// TwinCAT 3 PLC project main
// libraries:
//   Tc2_Math, * (Beckhoff Automation GmbH)
//   Tc2_MC2, * (Beckhoff Automation GmbH)
//   Tc2_Standard, * (Beckhoff Automation GmbH)
//   Tc2_System, * (Beckhoff Automation GmbH)
//   Tc3_Module, * (Beckhoff Automation GmbH)
//   VisuDialogs, * (System)
// project tree:
//   Global Variables/ Global_Variables.TcGVL, Variable_Configuration.TcGVL
//   / GlobalImagePool.TcGIPO (not stored), Standard.TcTTO, 视图管理器.TcVMO (not stored)
//   POUs/ AxisWriteParameter.TcPOU, Axis_Limit_Stop.TcPOU, Axis_Move.TcPOU, Axis_Power.TcPOU, Axis_stop.TcPOU, Axis_To_Zero.TcPOU, BackwardWindingStart.TcPOU, BLINK.TcPOU, ForwardWindingStart.TcPOU, MAIN.TcPOU, MainAxisRot.TcPOU, Manual_Left.TcPOU, Manual_Right.TcPOU, Motor_Init.TcPOU, Pulse2.TcPOU, ReadEncSpeed.TcPOU
//   Visualizations/ HMI1.TcVIS
// real-time tasks:
//   TASK Standard: cycle T#10ms, priority 20, ADS port 350
// motion (NC):
//   TASK NC-Task 1 SAF: cycle T#2ms, priority 4, ADS port 501
//   TASK NC-Task 1 SVB: cycle T#10ms, priority 8, ADS port 511
//   AXIS Axis 1 (id 1)
//     OtherSettings: AllowMotionCmdToSlave=true
//     encoder EncType=1
//       EncPara: ScaleFactorNumerator=0.00015625
//     drive DrvType=5
//       Analog: TorqueSetpointScale=10, ScaleFactorActTorque=0.1
//       TimeComp: TaskDelayCycles=1
//     controller CtrType=1
//       CtrPara: PriorControlFactor=1
//         Observer: BandWidth=20
//   AXIS Axis 2 (id 2)
//     OtherSettings: AllowMotionCmdToSlave=true
//     encoder EncType=4
//       EncPara: ScaleFactorNumerator=0.00025, MaxCount=#x0000ffff
//     drive DrvType=5
//       Analog: TorqueSetpointScale=10, ScaleFactorActTorque=0.1
//       TimeComp: TaskDelayCycles=1
//     controller CtrType=1
//       CtrPara: PriorControlFactor=1
//         Observer: BandWidth=20
//   AXIS Axis 3 (id 3)
//     OtherSettings: AllowMotionCmdToSlave=true
//     encoder EncType=1
//       EncPara: ScaleFactorNumerator=0.25
//     drive DrvType=5
//       Analog: TorqueSetpointScale=10, ScaleFactorActTorque=0.1
//       TimeComp: TaskDelayCycles=1
//     controller CtrType=1
//       CtrPara: PriorControlFactor=1
//         Observer: BandWidth=20
// variable links:
//   main/main Instance <-> NC-Task 1 SAF/Axes/Axis 1
//     Standard Inputs/.Axis1.NcToPlc <-> Outputs/ToPlc
//     Standard Outputs/.Axis1.PlcToNc <-> Inputs/FromPlc
//   main/main Instance <-> NC-Task 1 SAF/Axes/Axis 2
//     Standard Inputs/.Axis2.NcToPlc <-> Outputs/ToPlc
//     Standard Outputs/.Axis2.PlcToNc <-> Inputs/FromPlc
//   main/main Instance <-> NC-Task 1 SAF/Axes/Axis 3
//     Standard Inputs/.Axis3.NcToPlc <-> Outputs/ToPlc
//     Standard Outputs/.Axis3.PlcToNc <-> Inputs/FromPlc

CONFIGURATION main
    RESOURCE PLC ON TwinCAT3
        TASK Standard(INTERVAL := T#10ms, PRIORITY := 20);
        PROGRAM MAIN WITH Standard : MAIN;
    END_RESOURCE
END_CONFIGURATION

// ---- Global Variables/Global_Variables.TcGVL
{attribute 'Tc2GvlVarNames'}
VAR_GLOBAL
	Axis1: Axis_Ref;
	Axis2: Axis_Ref;
	Axis3: Axis_Ref;
END_VAR

// ---- Global Variables/Variable_Configuration.TcGVL
{attribute 'Tc2GvlVarNames'}
VAR_CONFIG
END_VAR

// ---- POUs/MAIN.TcPOU
PROGRAM MAIN
VAR_INPUT
	FootPedalPressed	AT%I*	:	BOOL;	(*主轴脚踏开关i1*)
	WireForwardWindingControl	AT%I*	:	BOOL;	(*自动排线正i2*)
	WireBackwardWindingControl	AT%I*	:	BOOL;	(*自动排线反i3*)
	MainAxisRotatingDirection AT%I*:	BOOL:= FALSE;	(*主轴旋转方向i4,TRUE 反向，FALSE正向*)
	MainAxisRotatingBackFlag: BOOL:= TRUE;
	cannel_5 AT%I*: BOOL;
	WireBackwardManualControl 	AT%I*	:	BOOL;	(*手动排线反i6*)
	WireForwardManualControl	AT%I*	:	BOOL;	(*手动排线正i7*)
	WireLeadPositiveLimit 	AT%I*	:	BOOL;	(*排线轴正限位i8*)
	WireLeadNegativeLimit 	AT%I*	:	BOOL;	(*排线轴负限位i9*)
	WireLeadToZero		AT%I*	:	BOOL;	(*排线轴寻零i10*)
	EL180911 AT%I*: BOOL;
	EL180912 AT%I*: BOOL;

	MainAxisSpeedControl	AT%I*	:	INT:=32767;		(*主轴调速, 模拟量*)

END_VAR
VAR_OUTPUT
	OpMode	AT%Q*: SINT:=8;	(*OP MODE*)
	Opmode2 AT%Q*: SINT:=8;	(*OP MODE*)

	status_Axis_forward		AT%Q*:	BOOL;	(*主轴正转o1*)
	status_Axis_backward		AT%Q*:	BOOL;	(*主轴反转o2*)
	Manual_control_forward	AT%Q*:	BOOL;	(*手动正转o3*)
	Manual_control_backward	AT%Q*:	BOOL;	(*手动反转o4*)
	Auto_control_forward		AT%Q*:	BOOL;	(*自动正转o5*)
	Auto_control_backward		AT%Q*:	BOOL;	(*自动反转o6*)
	Forward_position_limit		AT%Q*: 	BOOL;	(*起点限位o7*)
	Backward_position_limit	AT%Q*:	BOOL;	(*终点限位o8*)
	T510_X1		AT%Q*:	BOOL:=	FALSE;	(*T510的x1, 接主轴驱动器o9*)
	T510_X2		AT%Q*:	BOOL:=	FALSE;	(*T510的x2, 接主轴驱动器o10*)
	MotorEnable1 	AT%Q*:	BOOL:=	FALSE;	(*主轴电机使能o11*)
	MotorEnable2 	AT%Q*:	BOOL:=	FALSE;	(*主轴电机使能o12*)

END_VAR
VAR
	Flag1: BOOL;
	timer1: Pulse2;
	shanshuo: BLINK;

	AxisPower: Axis_Power;
	AxisReset2:MC_Reset;
	AxisReset1: MC_Reset;
	MoveVelPlus: MC_MoveVelocity;
	MoveVelDec: MC_MoveVelocity;
	absMove1: MC_MoveAbsolute;
	absMove2: MC_MoveAbsolute;

	MOTORINIT: Motor_Init;
	WriteParameter: AxisWriteParameter;
	AxisStop: Axis_Limit_Stop;
	AxisStop2: Axis_stop;
	AxisToZero:Axis_To_Zero;
	manleft:Manual_Left;
	manright			:	Manual_Right;
	AxisMove			:	Axis_Move;
	MainAxisRotation	:	MainAxisRot;
	ReadEncoderVel	:	ReadEncSpeed;
	WireWeights	:	REAL:=	2.4;
	TargetMainAxisSpeed	:	REAL:=	8;
	ManualControlVelocity	:	REAL:=	8;
	SlaveAxisBackZero	:	REAL:= 8;

END_VAR


(********************************************************  轴使能   ************************************************************)
AxisPower(
	SpeedControl:=MainAxisSpeedControl,
	Power_Status=> );
AxisReset1(
	Execute:=EL180911,
	Axis:= Axis1,
	Done=> ,
	Busy=> ,
	Error=> ,
	ErrorID=> );

AxisReset2(
	Execute:=EL180911,
	Axis:= Axis3,
	Done=> ,
	Busy=> ,
	Error=> ,
	ErrorID=> );

AxisStop(
	Execute_:=WireLeadPositiveLimit,
	Execute_2:=WireLeadNegativeLimit ,
	Decelerations:=1500,
	Flag1=>Forward_position_limit,
	Flag2=> Backward_position_limit);

ReadEncoderVel(input1:= AxisPower.Power_Status, RealSpeed=> );

(****************************************************  主轴旋转方向设定	********************************************************)
IF MainAxisRotatingDirection THEN
	MainAxisRotatingBackFlag:=FALSE;
	status_Axis_forward:=TRUE;
	status_Axis_backward:=FALSE;
ELSE
	MainAxisRotatingBackFlag:= TRUE;
	status_Axis_forward:=FALSE;
	status_Axis_backward:=TRUE;
END_IF

(******************************************************	正转向右启动	*******************************************************)
IF MainAxisRotatingDirection THEN
	IF FootPedalPressed THEN
			T510_X1:=TRUE;
			MOTORINIT(forward_start:=MainAxisRotatingDirection , backward_start:=T510_X1 , Flag=> MotorEnable1);
		ELSE
			T510_X1:=FALSE;
			MOTORINIT(forward_start:=FALSE , backward_start:=T510_X1 , Flag=> MotorEnable1);
	END_IF
	IF WireForwardWindingControl THEN
		IF FootPedalPressed THEN OpMode:=8;
		END_IF
	(*伺服动作*)
		MoveVelPlus(
				Execute:=FootPedalPressed ,
				Velocity:= (WireWeights*TargetMainAxisSpeed),
				Acceleration:= ,
				Deceleration:= ,
				Jerk:= ,
				Direction:= MC_Positive_Direction,
				BufferMode:= ,
				Options:= ,
				Axis:=Axis1 ,
				InVelocity=> ,
				Busy=> ,
				Active=>Auto_control_forward ,
				CommandAborted=> ,
				Error=> ,
				ErrorID=> );

		AxisStop2(Execute_:= FootPedalPressed);
		(*AxisMove(Input1:=FootPedalPressed );*)
	END_IF

	(*正向向左启动*)
	IF WireBackwardWindingControl THEN
		IF FootPedalPressed THEN OpMode:=8;
		END_IF
	(*私服动作*)
		MoveVelDec(
				Execute:= FootPedalPressed,
				Velocity:= (WireWeights*TargetMainAxisSpeed),
				Acceleration:= ,
				Deceleration:= ,
				Jerk:= ,
				Direction:= MC_Negative_Direction,
				BufferMode:= ,
				Options:= ,
				Axis:=Axis1 ,
				InVelocity=> ,
				Busy=> ,
				Active=>Auto_control_backward ,
				CommandAborted=> ,
				Error=> ,
				ErrorID=> );
		AxisStop2(Execute_:= FootPedalPressed);
	END_IF
END_IF


(*****************************************************	反转向右启动	******************************************************)
IF MainAxisRotatingBackFlag THEN
	IF FootPedalPressed THEN
			T510_X2:=TRUE;
			MOTORINIT(forward_start:=MainAxisRotatingBackFlag , backward_start:=T510_X2 , Flag=> MotorEnable1);
		ELSE
			T510_X2:=FALSE;
			MOTORINIT(
					forward_start:=FALSE ,
					backward_start:=T510_X2 ,
					Flag=> MotorEnable1);
	END_IF
	IF WireForwardWindingControl THEN
		IF FootPedalPressed THEN OpMode:=8;
		END_IF
		MoveVelPlus(
				Execute:=FootPedalPressed ,
				Velocity:= (WireWeights*TargetMainAxisSpeed),
				Acceleration:= ,
				Deceleration:= ,
				Jerk:= ,
				Direction:= MC_Positive_Direction,
				BufferMode:= ,
				Options:= ,
				Axis:=Axis1 ,
				InVelocity=> ,
				Busy=> ,
				Active=>Auto_control_forward ,
				CommandAborted=> ,
				Error=> ,
				ErrorID=> );
		AxisStop2(Execute_:= FootPedalPressed);
	END_IF

	(*反转向左启动*)
	IF WireBackwardWindingControl THEN
		MoveVelDec(
				Execute:= FootPedalPressed,
				Velocity:= (WireWeights*TargetMainAxisSpeed),
				Acceleration:= ,
				Deceleration:= ,
				Jerk:= ,
				Direction:= MC_Negative_Direction,
				BufferMode:= ,
				Options:= ,
				Axis:=Axis1 ,
				InVelocity=> ,
				Busy=> ,
				Active=>Auto_control_backward ,
				CommandAborted=> ,
				Error=> ,
				ErrorID=> );
		AxisStop2(Execute_:= FootPedalPressed);
	END_IF
END_IF


(*****************************************************	手动控制正向启动	************************************************************)
	(*私服动作*)
IF WireForwardManualControl THEN
	OpMode:=8;
END_IF
manleft(
	Input1:=	WireForwardManualControl,
	ManualCotrolSpeed	:=	ManualControlVelocity ,
	Flag1	=>	Manual_control_forward);

(*Flag1:=REAL_TO_INT(0.02432*MainAxisSpeedControl);
timer1(button1:= WireForwardManualControl, time_fuction:=Flag1, Flag=>status_Axis_forward );*)


(****************************************************	手动控制反向启动	************************************************************)
	(*私服动作*)
IF WireBackwardManualControl THEN
	OpMode:=8;
END_IF
manright(
	Input1:=WireBackwardManualControl,
	ManualCotrolSpeed	:=ManualControlVelocity ,
	Flag1=> Manual_control_backward);

(**********************************************************	排线轴归零	*********************************************************************)
IF WireLeadToZero THEN
	OpMode:=8;
END_IF
AxisToZero(
	Flag:= WireLeadToZero,
	BackZeroSpeed:=SlaveAxisBackZero);

(**********************************************************	主轴旋转控制	*****************************************************************)
IF FootPedalPressed THEN
	OpMode2:=8;
END_IF
MainAxisRotation(
	Input1:=FootPedalPressed,
	ForwardRotFlag:=MainAxisRotatingDirection,
	BackwardRotFlag:=MainAxisRotatingBackFlag,
	InputTargetSpeed:= TargetMainAxisSpeed);

END_PROGRAM

// ---- POUs/Pulse2.TcPOU
FUNCTION_BLOCK Pulse2
VAR_INPUT
	button1: BOOL;
	time_fuction: INT;
END_VAR
VAR_OUTPUT
	Flag: BOOL;
END_VAR
VAR
	Timer1: TON;
END_VAR

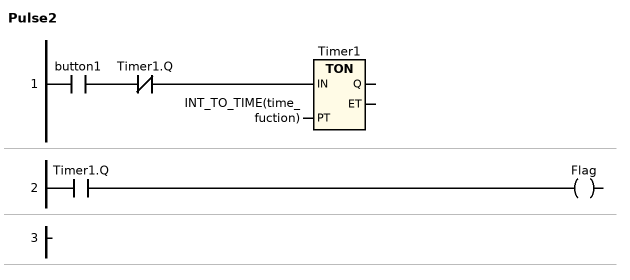
// NETWORK 1
Timer1(IN := button1 AND NOT Timer1.Q, PT := INT_TO_TIME(time_fuction)); // TON

// NETWORK 2
Flag := Timer1.Q;

// NETWORK 3

END_FUNCTION_BLOCK

// ---- POUs/BLINK.TcPOU
FUNCTION_BLOCK BLINK
VAR_INPUT
	ENABLE: BOOL;
END_VAR
VAR_OUTPUT
	OUT: BOOL;
END_VAR
VAR
	TIMELOW: INT;
	TIMEHIGH: INT;
	T37: TON;
	T38: TOF;
	TEMP1: BOOL;
END_VAR

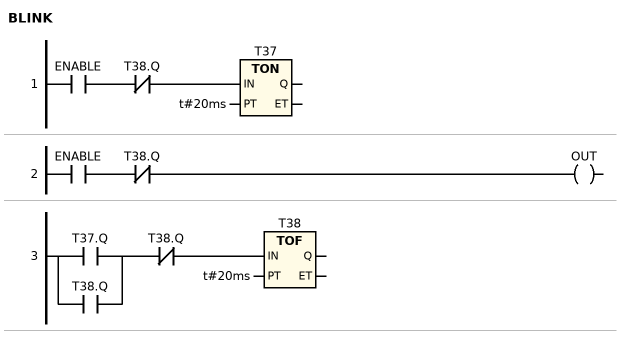
// NETWORK 1
T37(IN := ENABLE AND NOT T38.Q, PT := t#20ms); // TON

// NETWORK 2
OUT := ENABLE AND NOT T38.Q;

// NETWORK 3
T38(IN := (T37.Q OR T38.Q) AND NOT T38.Q, PT := t#20ms); // TOF

END_FUNCTION_BLOCK

// ---- POUs/Axis_Power.TcPOU
FUNCTION_BLOCK Axis_Power
VAR_INPUT
	SpeedControl:INT;
END_VAR
VAR_OUTPUT
	Power_Status:BOOL;
END_VAR
VAR
	AxisPower1: MC_Power;
	AxisPower2: MC_Power;
END_VAR

AxisPower1(
    Enable := TRUE,
    Enable_Positive := TRUE,
    Enable_Negative := TRUE,
    Override := REAL_TO_INT(0.00305185*SpeedControl),
    Axis := Axis1); // MC_Power
Power_Status := AxisPower1.Status;
AxisPower2(
    Enable := TRUE,
    Enable_Positive := TRUE,
    Enable_Negative := TRUE,
    Override := REAL_TO_INT(0.00305185*SpeedControl),
    Axis := Axis3); // MC_Power
Power_Status := AxisPower2.Status;

END_FUNCTION_BLOCK

// ---- POUs/Motor_Init.TcPOU
FUNCTION_BLOCK Motor_Init
VAR_INPUT
	forward_start: BOOL;
	backward_start: BOOL;
END_VAR
VAR_OUTPUT
	Flag: BOOL;
END_VAR

IF forward_start OR backward_start THEN
	Flag:=TRUE;
ELSE
	Flag:=FALSE;
END_IF

END_FUNCTION_BLOCK

// ---- POUs/AxisWriteParameter.TcPOU
FUNCTION_BLOCK AxisWriteParameter
VAR_INPUT
	Execute_:BOOL;
	Begin_Position:INT;
	End_Position:INT;
END_VAR
VAR_OUTPUT
END_VAR
VAR
	Write_Bool_Start	:	MC_WriteBoolParameter;
	Write_Bool_End 	:	MC_WriteBoolParameter;
	Write_Start :	MC_WriteParameter;
	Write_End :	MC_WriteParameter;
END_VAR

Write_Start(Execute := Execute_, ParameterNumber := 2, Value := End_Position, Axis := Axis1); // MC_WriteParameter
Write_End(Execute := Execute_, ParameterNumber := 3, Value := Begin_Position, Axis := Axis1); // MC_WriteParameter
Write_Bool_Start(Execute := Execute_, ParameterNumber := 4, Value := TRUE, Axis := Axis1); // MC_WriteBoolParameter
Write_Bool_End(Execute := Execute_, ParameterNumber := 5, Value := TRUE, Axis := Axis1); // MC_WriteBoolParameter

END_FUNCTION_BLOCK

// ---- POUs/Axis_Limit_Stop.TcPOU
FUNCTION_BLOCK Axis_Limit_Stop
VAR_INPUT
	Execute_:BOOL;
	Execute_2:BOOL;
	Decelerations: INT;
END_VAR
VAR_OUTPUT
	Flag1:BOOL;
	Flag2:BOOL;
END_VAR
VAR
	AxisStop:MC_Stop;
	trig1: F_TRIG;
END_VAR

AxisStop(Execute := Execute_ OR Execute_2, Deceleration := Decelerations, Axis := Axis1); // MC_Stop
Flag1 := Execute_;
Flag2 := Execute_2;

END_FUNCTION_BLOCK

// ---- POUs/Axis_stop.TcPOU
FUNCTION_BLOCK Axis_stop
VAR_INPUT
	Execute_:BOOL;
END_VAR
VAR_OUTPUT
END_VAR
VAR
	AxisStop:MC_Stop;
	trig1: F_TRIG;
END_VAR

trig1(CLK := Execute_); // F_TRIG
AxisStop(Execute := trig1.Q, Deceleration := 1500, Axis := Axis1); // MC_Stop

END_FUNCTION_BLOCK

// ---- POUs/Axis_To_Zero.TcPOU
FUNCTION_BLOCK Axis_To_Zero
VAR_INPUT
	Flag: BOOL;
	BackZeroSpeed	:	REAL;
END_VAR
VAR_OUTPUT
END_VAR
VAR
	AxisToZero: MC_MoveAbsolute;
END_VAR

AxisToZero(Execute := Flag, Position := 0, Velocity := BackZeroSpeed, Axis := Axis1); // MC_MoveAbsolute

END_FUNCTION_BLOCK

// ---- POUs/Manual_Left.TcPOU
FUNCTION_BLOCK Manual_Left
VAR_INPUT
	Input1:BOOL;
	ManualCotrolSpeed	:	REAL;
END_VAR
VAR_OUTPUT
	Flag1:BOOL;
END_VAR
VAR
	temp1:MC_MoveVelocity;
	AxisStop:MC_Stop;
	trig1: F_TRIG;
END_VAR

temp1(
    Execute := Input1,
    Velocity := ManualCotrolSpeed,
    Acceleration := 1500,
    Deceleration := 1500,
    Direction := MC_Positive_Direction,
    Axis := Axis1); // MC_MoveVelocity
trig1(CLK := temp1.InVelocity OR temp1.CommandAborted); // F_TRIG
AxisStop(Execute := trig1.Q, Deceleration := 1500, Axis := Axis1); // MC_Stop
Flag1 := temp1.Active;

END_FUNCTION_BLOCK

// ---- POUs/Manual_Right.TcPOU
FUNCTION_BLOCK Manual_Right
VAR_INPUT
	Input1:BOOL;
	ManualCotrolSpeed	:	REAL;
END_VAR
VAR_OUTPUT
	Flag1:BOOL;
END_VAR
VAR
	temp1:MC_MoveVelocity;
	AxisStop:MC_Stop;
	trig1: F_TRIG;
END_VAR
VAR // added by the converter: edge detectors and wires of the graphical bodies
    _w1 : ANY;
END_VAR

temp1(
    Execute := Input1,
    Velocity := ManualCotrolSpeed,
    Acceleration := 1500,
    Deceleration := 1500,
    Direction := MC_Negative_Direction,
    Axis := Axis1); // MC_MoveVelocity
trig1(CLK := _w1); // F_TRIG
AxisStop(Execute := trig1.Q, Deceleration := 1500, Axis := Axis1); // MC_Stop
_w1 := temp1.InVelocity OR temp1.CommandAborted;
Flag1 := temp1.Active;

END_FUNCTION_BLOCK

// ---- POUs/Axis_Move.TcPOU
FUNCTION_BLOCK Axis_Move
VAR_INPUT
	Input1:BOOL;
END_VAR
VAR_OUTPUT
END_VAR
VAR
	absMove1: MC_MoveAbsolute;
	absMove2: MC_MoveAbsolute;
	pulse1:R_TRIG;
	Pulse2:R_TRIG;
	Pulse3:R_TRIG;
	CTU1:CTU;
	AxisStop:MC_Stop;
	trig1: F_TRIG;

END_VAR

absMove1(
    Execute := Pulse2.Q OR pulse3.Q,
    Position := 210,
    Velocity := 100,
    Acceleration := 1500,
    Axis := Axis1); // MC_MoveAbsolute
absMove2(Execute := pulse1.Q, Position := 0, Velocity := 100, Axis := Axis1); // MC_MoveAbsolute
pulse1(CLK := absMove1.Done); // R_TRIG
Pulse2(CLK := absMove2.Done); // R_TRIG
AxisStop(Execute := trig1.Q, Deceleration := 1500, Axis := Axis1); // MC_Stop
pulse3(CLK := CTU1.Q); // R_TRIG
CTU1(CU := Input1, PV := 1); // CTU
trig1(CLK := Input1); // F_TRIG

END_FUNCTION_BLOCK

// ---- POUs/MainAxisRot.TcPOU
FUNCTION_BLOCK MainAxisRot
VAR_INPUT
	Input1:BOOL;
	InputTargetSpeed	:	REAL;
	ForwardRotFlag	:	BOOL;
	BackwardRotFlag	:	BOOL;
END_VAR
VAR_OUTPUT
END_VAR
VAR
	temp1, temp2 	:	MC_MoveVelocity;
	AxisStop	:	MC_Stop;
	trig1, trig2	: 	F_TRIG;
END_VAR
VAR // added by the converter: edge detectors and wires of the graphical bodies
    _w1, _w2 : ANY;
END_VAR

temp1(
    Execute := _w1,
    Velocity := InputTargetSpeed,
    Acceleration := 1500,
    Deceleration := 1500,
    Direction := MC_Positive_Direction,
    Axis := Axis3); // MC_MoveVelocity
_w2 := trig1.Q OR trig2.Q;
_w1 := Input1 AND BackwardRotFlag;
trig1(CLK := temp1.InVelocity OR temp1.CommandAborted); // F_TRIG
AxisStop(Execute := _w2, Deceleration := 1500, Axis := Axis3); // MC_Stop
temp2(
    Execute := Input1 AND ForwardRotFlag,
    Velocity := InputTargetSpeed,
    Acceleration := 1500,
    Deceleration := 1500,
    Direction := MC_Negative_Direction,
    Axis := Axis3); // MC_MoveVelocity
trig2(CLK := temp2.InVelocity OR temp2.CommandAborted); // F_TRIG

END_FUNCTION_BLOCK

// ---- POUs/ReadEncSpeed.TcPOU
FUNCTION_BLOCK ReadEncSpeed
VAR_INPUT
	input1:BOOL;
END_VAR
VAR_OUTPUT
	RealSpeed:REAL;
END_VAR
VAR
	ver1	:MC_ReadActualVelocity;
END_VAR

ver1(Enable := input1, Axis := Axis3); // MC_ReadActualVelocity
RealSpeed := ver1.ActualVelocity;

END_FUNCTION_BLOCK

// ---- POUs/BackwardWindingStart.TcPOU
FUNCTION_BLOCK BackwardWindingStart
VAR_INPUT
	FootPedalPressed:	BOOL;	(*主轴脚踏开关*)
	WireBackwardWindingControl:	BOOL;	(*自动排线正*)
END_VAR
VAR_OUTPUT
	X2: BOOL;	(*T510的x1*)(*接主轴驱动器*)
	Enable: BOOL;
END_VAR
VAR
	EngineX2: BOOL;
	EngineEnable: BOOL;
END_VAR

(*反向绕线启动*)
IF FootPedalPressed  THEN
	IF WireBackwardWindingControl THEN
		X2:=TRUE;
		Enable:=TRUE;
	END_IF
ELSE
	X2:=FALSE;
	Enable:=FALSE;
END_IF
EngineX2:=X2;
EngineEnable:=Enable;

END_FUNCTION_BLOCK

// ---- POUs/ForwardWindingStart.TcPOU
FUNCTION_BLOCK ForwardWindingStart
VAR_INPUT
	FootPedalPressed:	BOOL;	(*主轴脚踏开关*)
	WireForwardWindingControl:	BOOL;	(*自动排线正*)
END_VAR
VAR_OUTPUT
	X1: BOOL;	(*T510的x1*)(*接主轴驱动器*)
	Enable: BOOL;
END_VAR
VAR
	EngineX1: BOOL;
	EngineEnable: BOOL;
END_VAR

(*正向绕线启动*)
IF FootPedalPressed THEN
	IF WireForwardWindingControl  THEN
		X1:=TRUE;
		Enable:=TRUE;
	END_IF
ELSE
	X1:=FALSE;
	Enable:=FALSE;
END_IF
EngineX1:=X1;
EngineEnable:=Enable;

END_FUNCTION_BLOCK

// ---- Visualizations/HMI1.TcVIS
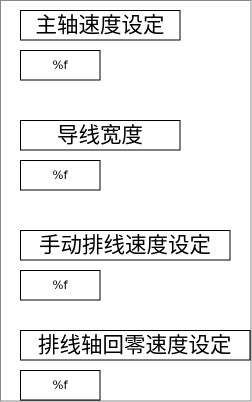
VISUALIZATION HMI1  // 252x402
    Rectangle (20,10 160x30), "主轴速度设定"
    Rectangle (20,50 80x30), "%f", text variable: MAIN.TargetMainAxisSpeed
        OnMouseDown: write the text variable via VisuDialogs.Numpad, min 0, max 20
    Rectangle (20,120 160x30), "导线宽度"
    Rectangle (20,230 210x30), "手动排线速度设定"
    Rectangle (20,330 230x30), "排线轴回零速度设定"
    Rectangle (20,160 80x30), "%f", text variable: MAIN.WireWeights
        OnMouseDown: write the text variable via VisuDialogs.Numpad, min 0, max 5
    Rectangle (20,270 80x30), "%f", text variable: MAIN.ManualControlVelocity
        OnMouseDown: write the text variable via VisuDialogs.Numpad, min 0, max 10
    Rectangle (20,370 80x30), "%f", text variable: MAIN.SlaveAxisBackZero
        OnMouseDown: write the text variable via VisuDialogs.Numpad, min 0, max 10
END_VISUALIZATION
